(* CoDeSys 2.3.9.59 project: main.pro *)
(* Libraries: TcBase.lib 14.5.09 12:14:08, TcSystem.lib 7.6.16 11:01:22, TcBaseMath.lib 27.7.04 12:07:56, TcMath.lib 23.9.04 15:15:30, TcMC2.lib 13.9.17 10:18:38, STANDARD.LIB *)

(* Task configuration *)
TASK Standard (PRIORITY := 0, INTERVAL := T#10ms);
	MAIN
END_TASK

(* Global variable list: Global_Variables *)
VAR_GLOBAL
	Axis1: Axis_Ref;
END_VAR

(* Global variable list: TwinCAT_Configuration *)
(* Generated automatically by TwinCAT - (read only) *)
VAR_CONFIG
	MAIN.FootPedalPressed AT %IX2.2 : BOOL;	(*  ~ {LinkedWith:TIID^Device 1 (EtherCAT)^Term 1 (EK1200)^Term 2 (EL1809)^Channel 1^Input} *)
	MAIN.WireForwardWindingControl AT %IX2.4 : BOOL;	(*  ~ {LinkedWith:TIID^Device 1 (EtherCAT)^Term 1 (EK1200)^Term 2 (EL1809)^Channel 2^Input} *)
	MAIN.WireBackwardWindingControl AT %IX2.5 : BOOL;	(*  ~ {LinkedWith:TIID^Device 1 (EtherCAT)^Term 1 (EK1200)^Term 2 (EL1809)^Channel 3^Input} *)
	MAIN.MainAxisRotatingDirection AT %IX2.3 : BOOL;	(*  ~ {LinkedWith:TIID^Device 1 (EtherCAT)^Term 1 (EK1200)^Term 2 (EL1809)^Channel 4^Input} *)
	MAIN.cannel_5 AT %IX3.3 : BOOL;	(*  ~ {LinkedWith:TIID^Device 1 (EtherCAT)^Term 1 (EK1200)^Term 2 (EL1809)^Channel 5^Input} *)
	MAIN.WireBackwardManualControl AT %IX2.7 : BOOL;	(*  ~ {LinkedWith:TIID^Device 1 (EtherCAT)^Term 1 (EK1200)^Term 2 (EL1809)^Channel 6^Input} *)
	MAIN.WireForwardManualControl AT %IX2.6 : BOOL;	(*  ~ {LinkedWith:TIID^Device 1 (EtherCAT)^Term 1 (EK1200)^Term 2 (EL1809)^Channel 7^Input} *)
	MAIN.WireLeadPositiveLimit AT %IX3.1 : BOOL;	(*  ~ {LinkedWith:TIID^Device 1 (EtherCAT)^Term 1 (EK1200)^Term 2 (EL1809)^Channel 8^Input} *)
	MAIN.WireLeadNegativeLimit AT %IX3.2 : BOOL;	(*  ~ {LinkedWith:TIID^Device 1 (EtherCAT)^Term 1 (EK1200)^Term 2 (EL1809)^Channel 9^Input} *)
	MAIN.WireLeadToZero AT %IX3.0 : BOOL;	(*  ~ {LinkedWith:TIID^Device 1 (EtherCAT)^Term 1 (EK1200)^Term 2 (EL1809)^Channel 10^Input} *)
	MAIN.EL180911 AT %IX2.0 : BOOL;	(*  ~ {LinkedWith:TIID^Device 1 (EtherCAT)^Term 1 (EK1200)^Term 2 (EL1809)^Channel 11^Input} *)
	MAIN.EL180912 AT %IB132 : UINT;	(*  ~ {LinkedWith:TIID^Device 1 (EtherCAT)^Term 1 (EK1200)^Term 6 (EL5101)^ENC Status compact^Counter value} *)
	MAIN.MainAxisSpeedControl AT %IB0 : INT;	(*  ~ {LinkedWith:TIID^Device 1 (EtherCAT)^Term 1 (EK1200)^Term 4 (EL3064)^AI Standard Channel 1^Value} *)
	MAIN.OpMode AT %QB132 : SINT;	(*  ~ {LinkedWith:TIID^Device 4 (EtherCAT)^Drive 8 (2DM556-EC)^RxPdoMapping^op_mode} *)
	MAIN.status_Axis_forward AT %QX133.1 : BOOL;	(*  ~ {LinkedWith:TIID^Device 1 (EtherCAT)^Term 1 (EK1200)^Term 3 (EL2809)^Channel 1^Output} *)
	MAIN.status_Axis_backward AT %QX133.2 : BOOL;	(*  ~ {LinkedWith:TIID^Device 1 (EtherCAT)^Term 1 (EK1200)^Term 3 (EL2809)^Channel 2^Output} *)
	MAIN.Manual_control_forward AT %QX133.3 : BOOL;	(*  ~ {LinkedWith:TIID^Device 1 (EtherCAT)^Term 1 (EK1200)^Term 3 (EL2809)^Channel 3^Output} *)
	MAIN.Manual_control_backward AT %QX133.4 : BOOL;	(*  ~ {LinkedWith:TIID^Device 1 (EtherCAT)^Term 1 (EK1200)^Term 3 (EL2809)^Channel 4^Output} *)
	MAIN.Auto_control_forward AT %QX133.5 : BOOL;	(*  ~ {LinkedWith:TIID^Device 1 (EtherCAT)^Term 1 (EK1200)^Term 3 (EL2809)^Channel 5^Output} *)
	MAIN.Auto_control_backward AT %QX133.6 : BOOL;	(*  ~ {LinkedWith:TIID^Device 1 (EtherCAT)^Term 1 (EK1200)^Term 3 (EL2809)^Channel 6^Output} *)
	MAIN.Forward_position_limit AT %QX133.7 : BOOL;	(*  ~ {LinkedWith:TIID^Device 1 (EtherCAT)^Term 1 (EK1200)^Term 3 (EL2809)^Channel 7^Output} *)
	MAIN.Backward_position_limit AT %QX134.0 : BOOL;	(*  ~ {LinkedWith:TIID^Device 1 (EtherCAT)^Term 1 (EK1200)^Term 3 (EL2809)^Channel 8^Output} *)
	MAIN.T510_X1 AT %QX0.1 : BOOL;	(*  ~ {LinkedWith:TIID^Device 1 (EtherCAT)^Term 1 (EK1200)^Term 3 (EL2809)^Channel 9^Output} *)
	MAIN.T510_X2 AT %QX0.0 : BOOL;	(*  ~ {LinkedWith:TIID^Device 1 (EtherCAT)^Term 1 (EK1200)^Term 3 (EL2809)^Channel 10^Output} *)
	MAIN.MotorEnable1 AT %QX0.2 : BOOL;	(*  ~ {LinkedWith:TIID^Device 1 (EtherCAT)^Term 1 (EK1200)^Term 3 (EL2809)^Channel 11^Output} *)
	MAIN.MotorEnable2 AT %QX0.3 : BOOL;	(*  ~ {LinkedWith:TIID^Device 1 (EtherCAT)^Term 1 (EK1200)^Term 3 (EL2809)^Channel 12^Output} *)
	.Axis1.PlcToNc AT %QB1 : PLCTONC_AXIS_REF;	(*  ~ {LinkedWith:TINC^NC-Task 1 SAF^Axes^ADM556^Inputs^ADM556_FromPlc} *)
	.Axis1.NcToPlc AT %IB4 : NCTOPLC_AXIS_REF;	(*  ~ {LinkedWith:TINC^NC-Task 1 SAF^Axes^ADM556^Outputs^ADM556_ToPlc} *)
END_VAR

(* POU MAIN, ST *)
PROGRAM MAIN
VAR_INPUT
	FootPedalPressed	AT%I*	:	BOOL;	(*主轴脚踏开关i1*)
	WireForwardWindingControl	AT%I*	:	BOOL;	(*自动排线正i2*)
	WireBackwardWindingControl	AT%I*	:	BOOL;	(*自动排线反i3*)
	MainAxisRotatingDirection AT%I*:	BOOL:= FALSE;	(*主轴旋转方向i4,TRUE 反向，FALSE正向*)
	MainAxisRotatingBackFlag: BOOL:= TRUE;
	cannel_5 AT%I*: BOOL;
	WireBackwardManualControl 	AT%I*	:	BOOL;	(*手动排线反i6*)
	WireForwardManualControl	AT%I*	:	BOOL;	(*手动排线正i7*)
	WireLeadPositiveLimit 	AT%I*	:	BOOL;	(*排线轴正限位i8*)
	WireLeadNegativeLimit 	AT%I*	:	BOOL;	(*排线轴负限位i9*)
	WireLeadToZero		AT%I*	:	BOOL;	(*排线轴寻零i10*)
	EL180911 AT%I*: BOOL;
	EL180912 AT%I*: UINT;

	MainAxisSpeedControl	AT%I*	:	INT;		(*主轴调速, 模拟量*)
END_VAR
VAR_OUTPUT
	OpMode	AT%Q*: SINT:=8;	(*OP MODE*)

	status_Axis_forward		AT%Q*:	BOOL;	(*主轴正转o1*)
	status_Axis_backward		AT%Q*:	BOOL;	(*主轴反转o2*)
	Manual_control_forward	AT%Q*:	BOOL;	(*手动正转o3*)
	Manual_control_backward	AT%Q*:	BOOL;	(*手动反转o4*)
	Auto_control_forward		AT%Q*:	BOOL;	(*自动正转o5*)
	Auto_control_backward		AT%Q*:	BOOL;	(*自动反转o6*)
	Forward_position_limit		AT%Q*: 	BOOL;	(*起点限位o7*)
	Backward_position_limit	AT%Q*:	BOOL;	(*终点限位o8*)
	T510_X1		AT%Q*:	BOOL:=	FALSE;	(*T510的x1, 接主轴驱动器o9*)
	T510_X2		AT%Q*:	BOOL:=	FALSE;	(*T510的x2, 接主轴驱动器o10*)
	MotorEnable1 	AT%Q*:	BOOL:=	FALSE;	(*主轴电机使能o11*)
	MotorEnable2 	AT%Q*:	BOOL:=	FALSE;	(*主轴电机使能o12*)

END_VAR
VAR
	Flag1: BOOL;
	timer1: Pulse2;
	MOTORINIT: Motor_Init;   (*???*)
	shanshuo: BLINK;

	AxisPower: Axis_Power;
	AxisReset:MC_Reset;
	WriteParameter: AxisWriteParameter;
	AxisStop: Axis_Limit_Stop;
	AxisStop2: Axis_stop;
	AxisReset1: MC_Reset;
	AxisToZero:Axis_To_Zero;
	MoveVelPlus: MC_MoveVelocity;
	MoveVelDec: MC_MoveVelocity;
	manleft:Manual_Left;
	manright:Manual_Right;
	AxisMove:Axis_Move;
	absMove1: MC_MoveAbsolute;
	absMove2: MC_MoveAbsolute;


END_VAR
(********************************************************  轴使能   ************************************************************)
AxisPower(
	SpeedControl:=MainAxisSpeedControl,
	Power_Status=> );
(*WriteParameter(
	Execute_:=AxisPower.Power_Status ,
	Begin_Position:= 0,
	End_Position:=210);*)
AxisReset1(
	Execute:=EL180911,
	Axis:= Axis1,
	Done=> ,
	Busy=> , 
	Error=> , 
	ErrorID=> );
AxisStop(
	Execute_:=WireLeadPositiveLimit,
	Execute_2:=WireLeadNegativeLimit ,
	Decelerations:=1500,
	Flag1=>Forward_position_limit,
	Flag2=> Backward_position_limit);


(****************************************************  主轴旋转方向设定	********************************************************)
IF MainAxisRotatingDirection THEN
	MainAxisRotatingBackFlag:=FALSE;
	status_Axis_forward:=TRUE;
	status_Axis_backward:=FALSE;
ELSE
	MainAxisRotatingBackFlag:= TRUE;
	status_Axis_forward:=FALSE;
	status_Axis_backward:=TRUE;
END_IF

(******************************************************	正转向右启动	*******************************************************)
IF MainAxisRotatingDirection THEN
	IF FootPedalPressed THEN
			T510_X1:=TRUE;
			MOTORINIT(forward_start:=MainAxisRotatingDirection , backward_start:=T510_X1 , Flag=> MotorEnable1);
		ELSE
			T510_X1:=FALSE;
			MOTORINIT(forward_start:=FALSE , backward_start:=T510_X1 , Flag=> MotorEnable1);
	END_IF
	IF WireForwardWindingControl THEN
		IF FootPedalPressed THEN OpMode:=8;
		END_IF
	(*伺服动作*)
		MoveVelPlus(
				Execute:=FootPedalPressed ,
				Velocity:= 60,
				Acceleration:= ,
				Deceleration:= ,
				Jerk:= ,
				Direction:= MC_Positive_Direction,
				BufferMode:= ,
				Options:= ,
				Axis:=Axis1 ,
				InVelocity=> ,
				Busy=> ,
				Active=>Auto_control_forward ,
				CommandAborted=> ,
				Error=> ,
				ErrorID=> );

		AxisStop2(Execute_:= FootPedalPressed);
		(*AxisMove(Input1:=FootPedalPressed );*)
	END_IF

	(*正向向左启动*)
	IF WireBackwardWindingControl THEN
		IF FootPedalPressed THEN OpMode:=8;
		END_IF
	(*私服动作*)
		MoveVelDec(
				Execute:= FootPedalPressed,
				Velocity:= 60,
				Acceleration:= ,
				Deceleration:= ,
				Jerk:= ,
				Direction:= MC_Negative_Direction,
				BufferMode:= ,
				Options:= ,
				Axis:=Axis1 ,
				InVelocity=> ,
				Busy=> ,
				Active=>Auto_control_backward ,
				CommandAborted=> ,
				Error=> ,
				ErrorID=> );
		AxisStop2(Execute_:= FootPedalPressed);
	END_IF
END_IF


(*****************************************************	反转向右启动	******************************************************)
IF MainAxisRotatingBackFlag THEN
	IF FootPedalPressed THEN
			T510_X2:=TRUE;
			MOTORINIT(forward_start:=MainAxisRotatingBackFlag , backward_start:=T510_X2 , Flag=> MotorEnable1);
		ELSE
			T510_X2:=FALSE;
			MOTORINIT(forward_start:=FALSE , backward_start:=T510_X2 , Flag=> MotorEnable1);
	END_IF
	IF WireForwardWindingControl THEN
		IF FootPedalPressed THEN OpMode:=8;
		END_IF
		MoveVelPlus(
				Execute:=FootPedalPressed ,
				Velocity:= 60,
				Acceleration:= ,
				Deceleration:= ,
				Jerk:= ,
				Direction:= MC_Positive_Direction,
				BufferMode:= ,
				Options:= ,
				Axis:=Axis1 ,
				InVelocity=> ,
				Busy=> ,
				Active=>Auto_control_forward ,
				CommandAborted=> ,
				Error=> ,
				ErrorID=> );
		AxisStop2(Execute_:= FootPedalPressed);
	END_IF

	(*反转向左启动*)
	IF WireBackwardWindingControl THEN
		MoveVelDec(
				Execute:= FootPedalPressed,
				Velocity:= 60,
				Acceleration:= ,
				Deceleration:= ,
				Jerk:= ,
				Direction:= MC_Negative_Direction,
				BufferMode:= ,
				Options:= ,
				Axis:=Axis1 ,
				InVelocity=> ,
				Busy=> ,
				Active=>Auto_control_backward ,
				CommandAborted=> ,
				Error=> ,
				ErrorID=> );
		AxisStop2(Execute_:= FootPedalPressed);
	END_IF
END_IF


EL180912;

(*****************************************************	手动控制正向启动	************************************************************)
	(*私服动作*)
IF WireForwardManualControl THEN
	OpMode:=8;END_IF
manleft(Input1:=WireForwardManualControl, Flag1=>Manual_control_forward);

(*Flag1:=REAL_TO_INT(0.02432*MainAxisSpeedControl);
timer1(button1:= WireForwardManualControl, time_fuction:=Flag1, Flag=>status_Axis_forward );*)


(****************************************************	手动控制反向启动	****************************************************************)
	(*私服动作*)
IF WireBackwardManualControl THEN
	OpMode:=8;END_IF
manright(Input1:=WireBackwardManualControl, Flag1=> Manual_control_backward);




(**********************************************************	排线轴归零	*********************************************************************)
IF WireLeadToZero THEN
	OpMode:=8;
	(*私服动作*)
END_IF
AxisToZero(Flag:= WireLeadToZero);


IF cannel_5 THEN
(*shanshuo(ENABLE:=cannel_5 , OUT=>status_Axis_backward )*);
END_IF
END_PROGRAM

(* POU Pulse2, LD *)
FUNCTION_BLOCK Pulse2
VAR_INPUT
	button1: BOOL;
	time_fuction: INT;
END_VAR
VAR_OUTPUT
	Flag: BOOL;
END_VAR
VAR
	Timer1: TON;
END_VAR
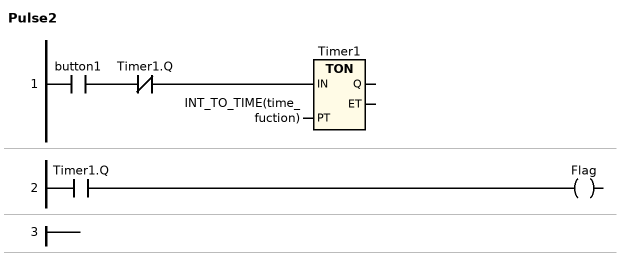
_LD_ (* Ladder Diagram *)
NETWORK 1
	[button1] - [/Timer1.Q] - Timer1:TON(IN: *, PT: INT_TO_TIME(time_fuction))
NETWORK 2
	[Timer1.Q] --- (Flag)
NETWORK 3
	*
_END_LD_
(* the same logic as Structured Text *)
(* Network 1 *)
Timer1(IN := button1 AND NOT Timer1.Q, PT := INT_TO_TIME(time_fuction));
(* Network 2 *)
Flag := Timer1.Q;
(* Network 3 *)
END_FUNCTION_BLOCK

(* POU Motor_Init, ST *)
FUNCTION_BLOCK Motor_Init
VAR_INPUT
	forward_start: BOOL;
	backward_start: BOOL;
END_VAR
VAR_OUTPUT
	Flag: BOOL;
END_VAR
IF forward_start OR backward_start THEN
	Flag:=TRUE;
ELSE
	Flag:=FALSE;
END_IF
END_FUNCTION_BLOCK

(* POU BLINK, LD *)
FUNCTION_BLOCK BLINK
VAR_INPUT
	ENABLE: BOOL;
END_VAR
VAR_OUTPUT
	OUT: BOOL;
END_VAR
VAR
	TIMELOW: INT;
	TIMEHIGH: INT;
	T37: TON;
	T38: TOF;
	TEMP1: BOOL;
END_VAR
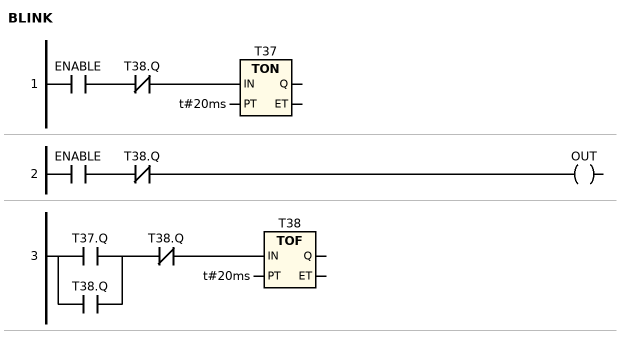
_LD_ (* Ladder Diagram *)
NETWORK 1
	[ENABLE] - [/T38.Q] - T37:TON(IN: *, PT: t#20ms)
NETWORK 2
	[ENABLE] - [/T38.Q] --- (OUT)
NETWORK 3
	{ [T37.Q] | [T38.Q] } - [/T38.Q] - T38:TOF(IN: *, PT: t#20ms)
_END_LD_
(* the same logic as Structured Text *)
(* Network 1 *)
T37(IN := ENABLE AND NOT T38.Q, PT := t#20ms);
(* Network 2 *)
OUT := ENABLE AND NOT T38.Q;
(* Network 3 *)
T38(IN := (T37.Q OR T38.Q) AND NOT T38.Q, PT := t#20ms);
END_FUNCTION_BLOCK

(* POU Axis_Power, CFC *)
FUNCTION_BLOCK Axis_Power
VAR_INPUT
	SpeedControl:INT;
END_VAR
VAR_OUTPUT
	Power_Status:BOOL;
END_VAR
VAR
	AxisPower: MC_Power;
END_VAR
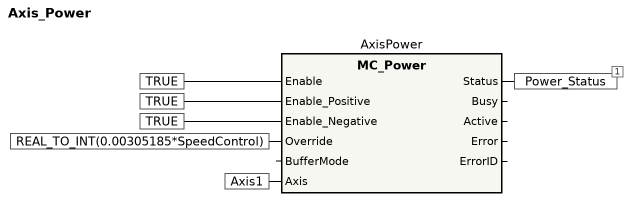
_CFC_ (* Continuous Function Chart, elements in execution order *)
#0 AxisPower:MC_Power(Enable: TRUE, Enable_Positive: TRUE, Enable_Negative: TRUE, Override: REAL_TO_INT(0.00305185*SpeedControl), BufferMode: -, Axis: Axis1)
#1 Power_Status <= #0.Status
_END_CFC_
(* the same logic as Structured Text *)
AxisPower(Enable := TRUE, Enable_Positive := TRUE, Enable_Negative := TRUE, Override := REAL_TO_INT(0.00305185*SpeedControl), Axis := Axis1);
Power_Status := AxisPower.Status;
END_FUNCTION_BLOCK

(* POU AxisWriteParameter, CFC *)
FUNCTION_BLOCK AxisWriteParameter
VAR_INPUT
	Execute_:BOOL;
	Begin_Position:INT;
	End_Position:INT;
END_VAR
VAR_OUTPUT
END_VAR
VAR
	Write_Bool_Start	:	MC_WriteBoolParameter;
	Write_Bool_End 	:	MC_WriteBoolParameter;
	Write_Start :	MC_WriteParameter;
	Write_End :	MC_WriteParameter;
END_VAR
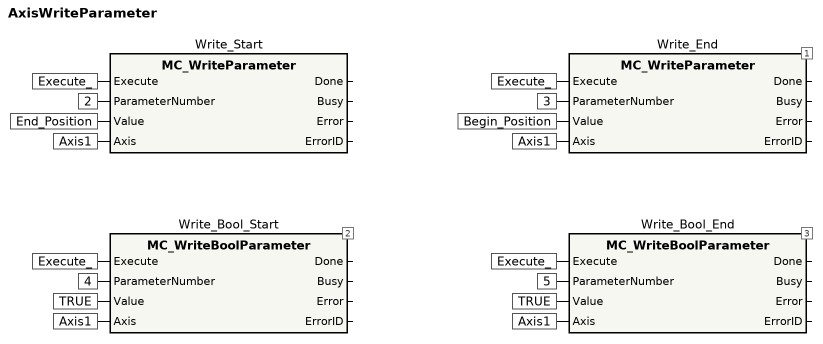
_CFC_ (* Continuous Function Chart, elements in execution order *)
#0 Write_Start:MC_WriteParameter(Execute: Execute_, ParameterNumber: 2, Value: End_Position, Axis: Axis1)
#1 Write_End:MC_WriteParameter(Execute: Execute_, ParameterNumber: 3, Value: Begin_Position, Axis: Axis1)
#2 Write_Bool_Start:MC_WriteBoolParameter(Execute: Execute_, ParameterNumber: 4, Value: TRUE, Axis: Axis1)
#3 Write_Bool_End:MC_WriteBoolParameter(Execute: Execute_, ParameterNumber: 5, Value: TRUE, Axis: Axis1)
_END_CFC_
(* the same logic as Structured Text *)
Write_Start(Execute := Execute_, ParameterNumber := 2, Value := End_Position, Axis := Axis1);
Write_End(Execute := Execute_, ParameterNumber := 3, Value := Begin_Position, Axis := Axis1);
Write_Bool_Start(Execute := Execute_, ParameterNumber := 4, Value := TRUE, Axis := Axis1);
Write_Bool_End(Execute := Execute_, ParameterNumber := 5, Value := TRUE, Axis := Axis1);
END_FUNCTION_BLOCK

(* POU Axis_Limit_Stop, CFC *)
FUNCTION_BLOCK Axis_Limit_Stop
VAR_INPUT
	Execute_:BOOL;
	Execute_2:BOOL;
	Decelerations: INT;
END_VAR
VAR_OUTPUT
	Flag1:BOOL;
	Flag2:BOOL;
END_VAR
VAR
	AxisStop:MC_Stop;
	trig1: F_TRIG;
END_VAR
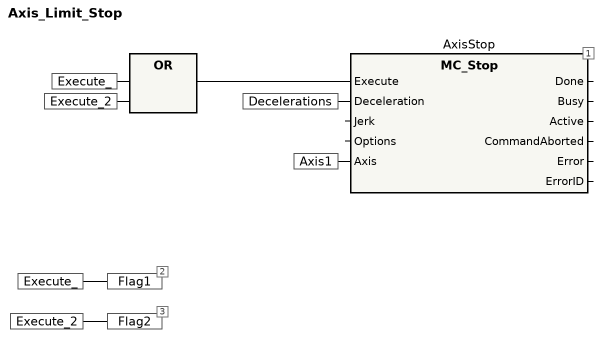
_CFC_ (* Continuous Function Chart, elements in execution order *)
#0 OR(Execute_, Execute_2)
#1 AxisStop:MC_Stop(Execute: #0, Deceleration: Decelerations, Jerk: -, Options: -, Axis: Axis1)
#2 Flag1 <= Execute_
#3 Flag2 <= Execute_2
_END_CFC_
(* the same logic as Structured Text *)
AxisStop(Execute := Execute_ OR Execute_2, Deceleration := Decelerations, Axis := Axis1);
Flag1 := Execute_;
Flag2 := Execute_2;
END_FUNCTION_BLOCK

(* POU Axis_stop, CFC *)
FUNCTION_BLOCK Axis_stop
VAR_INPUT
	Execute_:BOOL;
END_VAR
VAR_OUTPUT
END_VAR
VAR
	AxisStop:MC_Stop;
	trig1: F_TRIG;
END_VAR
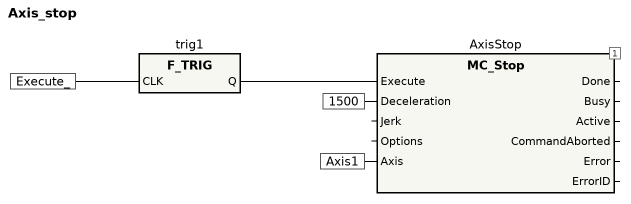
_CFC_ (* Continuous Function Chart, elements in execution order *)
#0 trig1:F_TRIG(CLK: Execute_)
#1 AxisStop:MC_Stop(Execute: #0.Q, Deceleration: 1500, Jerk: -, Options: -, Axis: Axis1)
_END_CFC_
(* the same logic as Structured Text *)
trig1(CLK := Execute_);
AxisStop(Execute := trig1.Q, Deceleration := 1500, Axis := Axis1);
END_FUNCTION_BLOCK

(* POU Axis_To_Zero, CFC *)
FUNCTION_BLOCK Axis_To_Zero
VAR_INPUT
	Flag: BOOL;
END_VAR
VAR_OUTPUT
END_VAR
VAR
	AxisToZero: MC_MoveAbsolute;
END_VAR
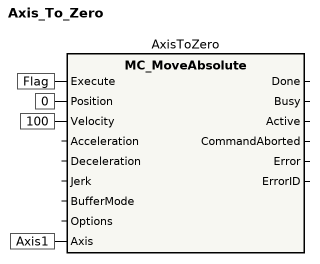
_CFC_ (* Continuous Function Chart, elements in execution order *)
#0 AxisToZero:MC_MoveAbsolute(Execute: Flag, Position: 0, Velocity: 100, Acceleration: -, Deceleration: -, Jerk: -, BufferMode: -, Options: -, Axis: Axis1)
_END_CFC_
(* the same logic as Structured Text *)
AxisToZero(Execute := Flag, Position := 0, Velocity := 100, Axis := Axis1);
END_FUNCTION_BLOCK

(* POU Manual_Left, CFC *)
FUNCTION_BLOCK Manual_Left
VAR_INPUT
	Input1:BOOL;
END_VAR
VAR_OUTPUT
	Flag1:BOOL;
END_VAR
VAR
	temp1:MC_MoveVelocity;
	AxisStop:MC_Stop;
	trig1: F_TRIG;
END_VAR
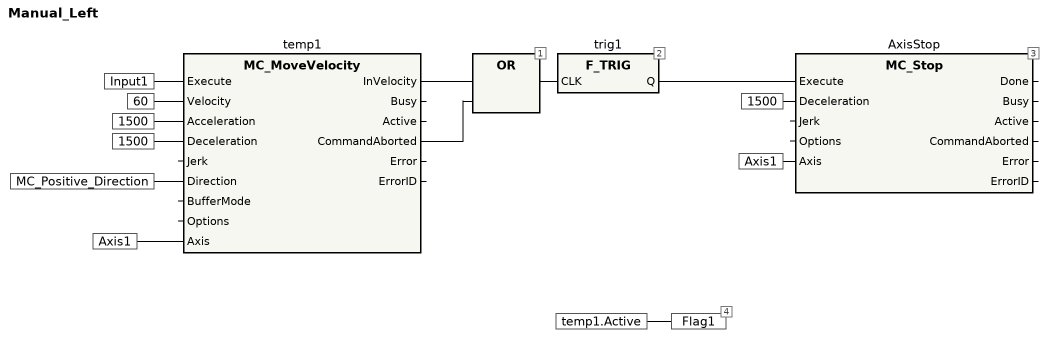
_CFC_ (* Continuous Function Chart, elements in execution order *)
#0 temp1:MC_MoveVelocity(Execute: Input1, Velocity: 60, Acceleration: 1500, Deceleration: 1500, Jerk: -, Direction: MC_Positive_Direction, BufferMode: -, Options: -, Axis: Axis1)
#1 OR(#0.InVelocity, #0.CommandAborted)
#2 trig1:F_TRIG(CLK: #1)
#3 AxisStop:MC_Stop(Execute: #2.Q, Deceleration: 1500, Jerk: -, Options: -, Axis: Axis1)
#4 Flag1 <= temp1.Active
_END_CFC_
(* the same logic as Structured Text *)
temp1(Execute := Input1, Velocity := 60, Acceleration := 1500, Deceleration := 1500, Direction := MC_Positive_Direction, Axis := Axis1);
trig1(CLK := temp1.InVelocity OR temp1.CommandAborted);
AxisStop(Execute := trig1.Q, Deceleration := 1500, Axis := Axis1);
Flag1 := temp1.Active;
END_FUNCTION_BLOCK

(* POU Manual_Right, CFC *)
FUNCTION_BLOCK Manual_Right
VAR_INPUT
	Input1:BOOL;
END_VAR
VAR_OUTPUT
	Flag1:BOOL;
END_VAR
VAR
	temp1:MC_MoveVelocity;
	AxisStop:MC_Stop;
	trig1: F_TRIG;
END_VAR
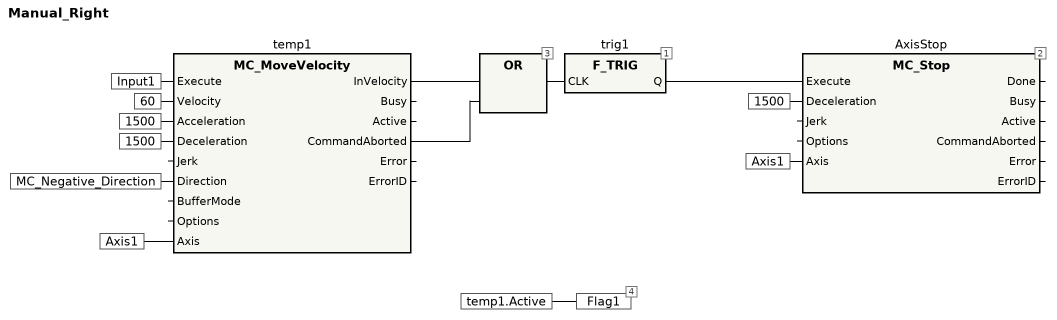
_CFC_ (* Continuous Function Chart, elements in execution order *)
#0 temp1:MC_MoveVelocity(Execute: Input1, Velocity: 60, Acceleration: 1500, Deceleration: 1500, Jerk: -, Direction: MC_Negative_Direction, BufferMode: -, Options: -, Axis: Axis1)
#1 trig1:F_TRIG(CLK: #3)
#2 AxisStop:MC_Stop(Execute: #1.Q, Deceleration: 1500, Jerk: -, Options: -, Axis: Axis1)
#3 OR(#0.InVelocity, #0.CommandAborted)
#4 Flag1 <= temp1.Active
_END_CFC_
END_FUNCTION_BLOCK

(* POU Axis_Move, CFC *)
FUNCTION_BLOCK Axis_Move
VAR_INPUT
	Input1:BOOL;
END_VAR
VAR_OUTPUT
END_VAR
VAR
	absMove1: MC_MoveAbsolute;
	absMove2: MC_MoveAbsolute;
	pulse1:R_TRIG;
	Pulse2:R_TRIG;
	Pulse3:R_TRIG;
	CTU1:CTU;
	AxisStop:MC_Stop;
	trig1: F_TRIG;

END_VAR
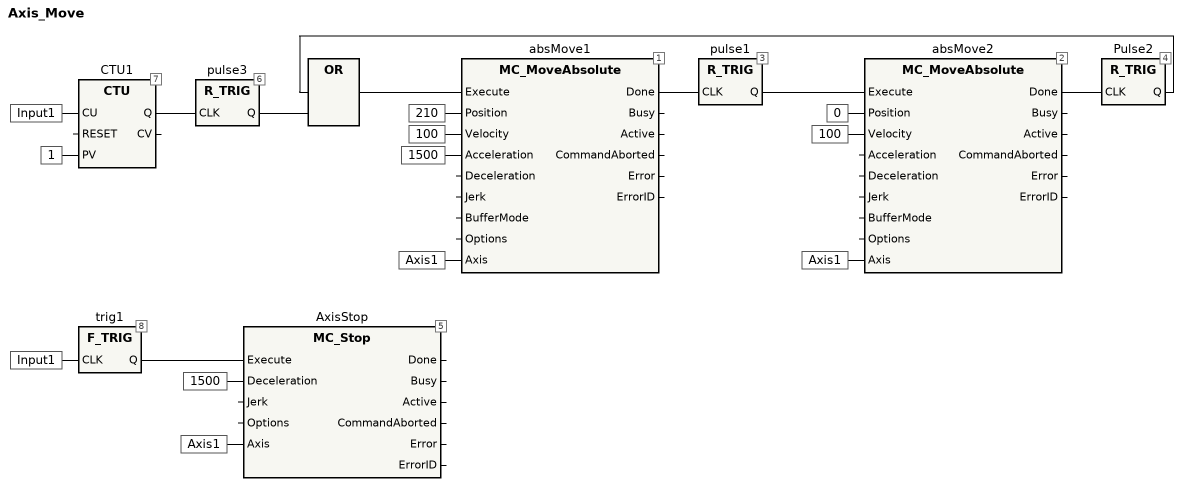
_CFC_ (* Continuous Function Chart, elements in execution order *)
#0 OR(#4.Q, #6.Q)
#1 absMove1:MC_MoveAbsolute(Execute: #0, Position: 210, Velocity: 100, Acceleration: 1500, Deceleration: -, Jerk: -, BufferMode: -, Options: -, Axis: Axis1)
#2 absMove2:MC_MoveAbsolute(Execute: #3.Q, Position: 0, Velocity: 100, Acceleration: -, Deceleration: -, Jerk: -, BufferMode: -, Options: -, Axis: Axis1)
#3 pulse1:R_TRIG(CLK: #1.Done)
#4 Pulse2:R_TRIG(CLK: #2.Done)
#5 AxisStop:MC_Stop(Execute: #8.Q, Deceleration: 1500, Jerk: -, Options: -, Axis: Axis1)
#6 pulse3:R_TRIG(CLK: #7.Q)
#7 CTU1:CTU(CU: Input1, RESET: -, PV: 1)
#8 trig1:F_TRIG(CLK: Input1)
_END_CFC_
(* the same logic as Structured Text *)
absMove1(Execute := Pulse2.Q OR pulse3.Q, Position := 210, Velocity := 100, Acceleration := 1500, Axis := Axis1);
absMove2(Execute := pulse1.Q, Position := 0, Velocity := 100, Axis := Axis1);
pulse1(CLK := absMove1.Done);
Pulse2(CLK := absMove2.Done);
AxisStop(Execute := trig1.Q, Deceleration := 1500, Axis := Axis1);
pulse3(CLK := CTU1.Q);
CTU1(CU := Input1, PV := 1);
trig1(CLK := Input1);
END_FUNCTION_BLOCK

(* POU BackwardWindingStart, ST *)
FUNCTION_BLOCK BackwardWindingStart
VAR_INPUT
	FootPedalPressed:	BOOL;	(*主轴脚踏开关*)
	WireBackwardWindingControl:	BOOL;	(*自动排线正*)
END_VAR
VAR_OUTPUT
	X2: BOOL;	(*T510的x1*)(*接主轴驱动器*)
	Enable: BOOL;
END_VAR
VAR
	EngineX2: BOOL;
	EngineEnable: BOOL;
END_VAR
(*反向绕线启动*)
IF FootPedalPressed  THEN
	IF WireBackwardWindingControl THEN
		X2:=TRUE;
		Enable:=TRUE;
	END_IF
ELSE
	X2:=FALSE;
	Enable:=FALSE;
END_IF
EngineX2:=X2;
EngineEnable:=Enable;
END_FUNCTION_BLOCK

(* POU ForwardWindingStart, ST *)
FUNCTION_BLOCK ForwardWindingStart
VAR_INPUT
	FootPedalPressed:	BOOL;	(*主轴脚踏开关*)
	WireForwardWindingControl:	BOOL;	(*自动排线正*)
END_VAR
VAR_OUTPUT
	X1: BOOL;	(*T510的x1*)(*接主轴驱动器*)
	Enable: BOOL;
END_VAR
VAR
	EngineX1: BOOL;
	EngineEnable: BOOL;
END_VAR
(*正向绕线启动*)
IF FootPedalPressed THEN
	IF WireForwardWindingControl  THEN
		X1:=TRUE;
		Enable:=TRUE;
	END_IF
ELSE
	X1:=FALSE;
	Enable:=FALSE;
END_IF
EngineX1:=X1;
EngineEnable:=Enable;
END_FUNCTION_BLOCK
